(* Schneider Machine Expert - Basic project pembuatn_makanan_otomatis(incomplete), file version 2.7.0.0 *)
(* ProjectInformations: Name=New project *)

HARDWARE
  Cpu 0: TM221M16R/G
  EthernetConfiguration: NetworkName=M221, IpAllocationMode=FixedAddress, IpAddress=0.0.0.0, SubnetMask=0.0.0.0
  SerialLineConfiguration: Baud=Baud19200, Parity=ParityEven, DataBits=DataBits8, StopBits=StopBits1, PhysicalMedium=PhysicalMediumRs485, TransmissionMode=TransmissionModeModbusRtu, SlaveId=1, Addressing=SlaveAddressing
  MastTask: UsePeriodScanMode=false, PeriodScan=100
  FastTask: Period=255
  CpuBehavior: StartingMode=StartAsPreviousState, AutoSaveRamOnEeprom=true, WatchdogPeriod=250

SYMBOLS  (address, symbol, comment, settings)
  %M0       IS_TARTED
  %I0.0     STARTING
  %I0.1     STOP

POU New POU
  (* SectionNumber=0 *)

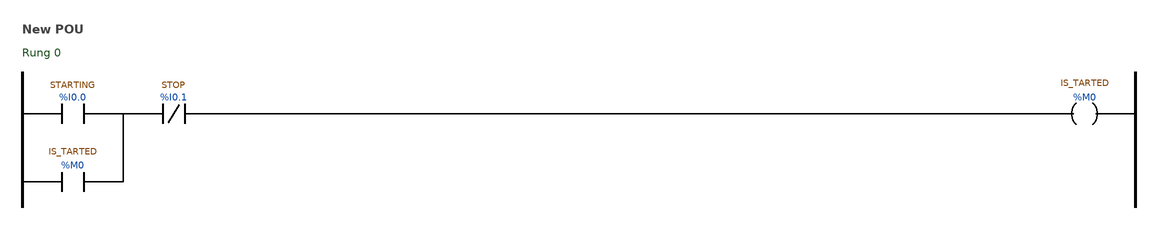

// Rung 0
  LD %I0.0                (* STARTING *)
  OR %M0                  (* IS_TARTED *)
  ANDN %I0.1              (* STOP *)
  ST %M0                  (* IS_TARTED *)
  // as ST:
  //   IS_TARTED := (STARTING OR IS_TARTED) AND NOT STOP;
